TYPE U_NCI_INDEX_GROUP :
UNION

  stCtrl              : ARRAY[1..MAX_NCI_CH] OF ST_Index_Group;

  byCtrl    AT %q*    : ARRAY[1..MAX_NCI_CH] OF
                        ARRAY[1..SIZEOF(ST_Index_Group)] OF BYTE;
END_UNION
END_TYPE

(* stored: Version 1.1.0.1
   DUT U_NCI_INDEX_GROUP: Id {7287b85b-33a4-4a5a-b2f8-d06fe82afead} *)
